PROGRAM Axe_04_Y_Laser	
VAR	YLaser:FB_Axe_Ethercat_V3;		Dem_gv_Y1,	B_Reset_Y1:BOOL;		TP_not_machine_en_service: TP;
	ACompleter_Y_decoupe_en_cours: BOOL;
END_VAR

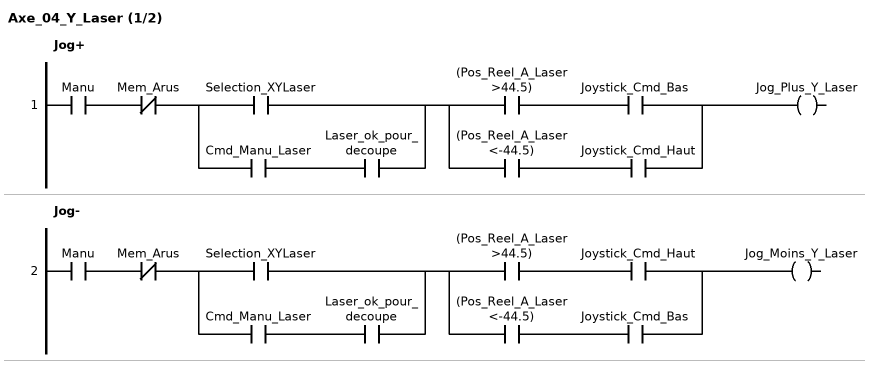
// NETWORK 1: Jog+
Jog_Plus_Y_Laser := Manu AND NOT Mem_Arus AND (Selection_XYLaser OR Cmd_Manu_Laser AND Laser_ok_pour_decoupe) AND (((Pos_Reel_A_Laser >44.5)) AND Joystick_Cmd_Bas OR ((Pos_Reel_A_Laser <-44.5)) AND Joystick_Cmd_Haut);

// NETWORK 2: Jog-
Jog_Moins_Y_Laser := Manu AND NOT Mem_Arus AND (Selection_XYLaser OR Cmd_Manu_Laser AND Laser_ok_pour_decoupe) AND (((Pos_Reel_A_Laser >44.5)) AND Joystick_Cmd_Haut OR ((Pos_Reel_A_Laser <-44.5)) AND Joystick_Cmd_Bas);

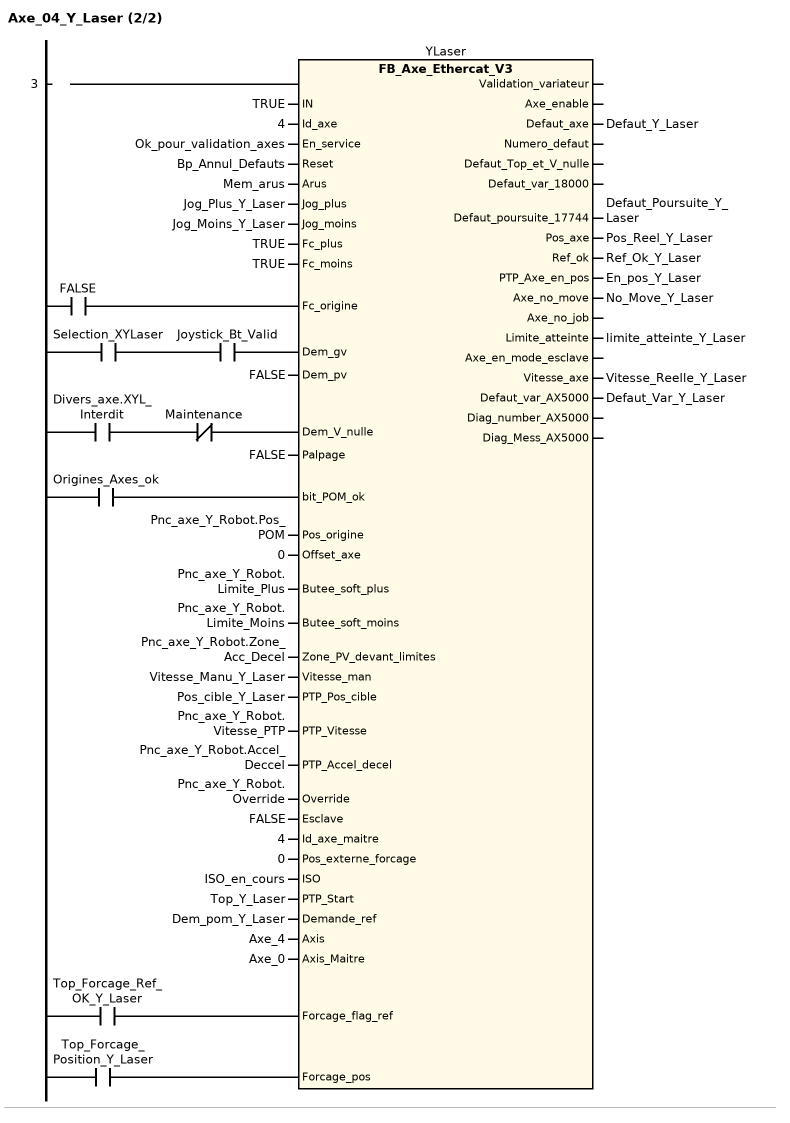
// NETWORK 3
//   Pnc_axe_Y_Robot.Pos_POM: 14
//   Pnc_axe_Y_Robot.Zone_Acc_Decel: 10
//   Pos_cible_Y_Laser: Axe Y Superieur
//   Pnc_axe_Y_Robot.Accel_Deccel: 6
//   Pnc_axe_Y_Robot.Override: 7
//   Axe_4: ***************************** Variables Axe3---Y1 *****************************
//   Axe_0: Axe bidon mais nécessaire car il est obligatoire de lier un axe maître en entrée de chaque FB_axe
YLaser(
    IN := TRUE,
    Id_axe := 4,
    En_service := Ok_pour_validation_axes,
    Reset := Bp_Annul_Defauts,
    Arus := Mem_arus,
    Jog_plus := Jog_Plus_Y_Laser,
    Jog_moins := Jog_Moins_Y_Laser,
    Fc_plus := TRUE,
    Fc_moins := TRUE,
    Fc_origine := FALSE,
    Dem_gv := Selection_XYLaser AND Joystick_Bt_Valid,
    Dem_pv := FALSE,
    Dem_V_nulle := Divers_axe.XYL_Interdit AND NOT Maintenance,
    Palpage := FALSE,
    bit_POM_ok := Origines_Axes_ok,
    Pos_origine := Pnc_axe_Y_Robot.Pos_POM,
    Offset_axe := 0,
    Butee_soft_plus := Pnc_axe_Y_Robot.Limite_Plus,
    Butee_soft_moins := Pnc_axe_Y_Robot.Limite_Moins,
    Zone_PV_devant_limites := Pnc_axe_Y_Robot.Zone_Acc_Decel,
    Vitesse_man := Vitesse_Manu_Y_Laser,
    PTP_Pos_cible := Pos_cible_Y_Laser,
    PTP_Vitesse := Pnc_axe_Y_Robot.Vitesse_PTP,
    PTP_Accel_decel := Pnc_axe_Y_Robot.Accel_Deccel,
    Override := Pnc_axe_Y_Robot.Override,
    Esclave := FALSE,
    Id_axe_maitre := 4,
    Pos_externe_forcage := 0,
    ISO := ISO_en_cours,
    PTP_Start := Top_Y_Laser,
    Demande_ref := Dem_pom_Y_Laser,
    Axis := Axe_4,
    Axis_Maitre := Axe_0,
    Forcage_flag_ref := Top_Forcage_Ref_OK_Y_Laser,
    Forcage_pos := Top_Forcage_Position_Y_Laser,
    Defaut_axe => Defaut_Y_Laser,
    Defaut_poursuite_17744 => Defaut_Poursuite_Y_Laser,
    Pos_axe => Pos_Reel_Y_Laser,
    Ref_ok => Ref_Ok_Y_Laser,
    PTP_Axe_en_pos => En_pos_Y_Laser,
    Axe_no_move => No_Move_Y_Laser,
    Limite_atteinte => limite_atteinte_Y_Laser,
    Vitesse_axe => Vitesse_Reelle_Y_Laser,
    Defaut_var_AX5000 => Defaut_Var_Y_Laser); // FB_Axe_Ethercat_V3

END_PROGRAM

(* stored: Version 1.1.0.1
   POU Axe_04_Y_Laser: Id {58275680-a780-431b-b840-09020c21657e}, SpecialFunc None *)
